//Structure is a mechanism of incubating divverent types under one logical name
TYPE myPersonType :
STRUCT
	name:STRING;
	age:INT;
	gendre:myGenderType;//unknown:=0,male:=1,female:=2
END_STRUCT
END_TYPE

(* stored: Version 1.1.0.1, ProductVersion 3.1.4024.11
   DUT myPersonType: Id {5f778bbc-a30a-4e82-bb39-5039cb3b7d3d} *)
